# EPICS autosave request: ip/ipApp/Db/CPSyringe_settings.req
# CPSyringe_settings.req
#
# Autosave file for Cole-Palmer Syringe Pump
#
# Mark Rivers
# November 23, 2013

$(P)$(R)ReadSettings.SCAN
$(P)$(R)Mode
$(P)$(R)Diameter
$(P)$(R)InfusionRate
$(P)$(R)InfusionRate.EGU
$(P)$(R)WithdrawalRate
$(P)$(R)WithdrawalRate.EGU
$(P)$(R)InfusionVolume
$(P)$(R)InfusionVolume.EGU
$(P)$(R)WithdrawalVolume
$(P)$(R)WithdrawalVolume.EGU
